FUNCTION_BLOCK ProcessBlock
VAR_INPUT
	ixIncPos: BOOL ;
	ixDecPos: BOOL;
END_VAR
VAR_OUTPUT
	PosValue: UINT := 0;
END_VAR
VAR
END_VAR


IF GVL.ixButtManual OR GVL.ixButtAuto THEN
	IF ixIncPos AND PosValue <= 900 AND NOT GVL.qxSensor2 THEN
		IF PosValue > 895 AND PosValue < 900 THEN
			PosValue := 900;
		ELSIF PosValue <= 895 THEN
			PosValue := PosValue + 5;
		END_IF
	END_IF

	IF ixDecPos AND PosValue >= 0 AND NOT GVL.qxSensor1 THEN
		IF PosValue < 5 AND PosValue > 0 THEN
			PosValue := 0;
		ELSIF PosValue >= 5 THEN
			PosValue := PosValue - 5;
		END_IF
	END_IF
END_IF

END_FUNCTION_BLOCK

(* stored: Version 1.1.0.1, ProductVersion 3.1.4024.12
   POU ProcessBlock: Id {d5a82c08-2d96-41c2-b237-9a8ed9e22122}, SpecialFunc None *)
